{attribute addProperty BoxType "KL1382"}
{attribute addProperty Id "Channel_1Channel_3D8C2EB100Channel_2Channel_3D8C2EB100"}
{attribute addProperty CRC "2978215931"}
{attribute addProperty SizeInBites "0"}
{attribute addProperty SizeInBytes "0"}
TYPE KL1382_B183F7FB :
STRUCT
	{attribute addProperty Name "Channel_1"}
	Channel_1 : Channel_3D8C2EB1;
	{attribute addProperty Name "Channel_2"}
	Channel_2 : Channel_3D8C2EB1;
END_STRUCT
END_TYPE

(* stored: Version 1.2.0.0, ProductVersion 3.1.4024.9
   DUT KL1382_B183F7FB: Id {5b1a07e8-ddf8-457a-aef3-f03ea1757578} *)
